% RSLogix 500 project TOFF Que 3.RSS, saved by version 8.30.00.15 %
PROJECT "UNTITLED"    % processor: MicroLogix 1400 %

PROGRAM FILES
  LAD 2   5 rungs

DATA FILES
  O0 OUTPUT  6 elements
  I1 INPUT  8 elements
  S2 STATUS  66 elements
  B3 BINARY  1 elements
  T4 TIMER  3 elements
  C5 COUNTER  1 elements
  R6 CONTROL  1 elements
  N7 INTEGER  1 elements
  F8 FLOAT  1 elements

LADDER 2
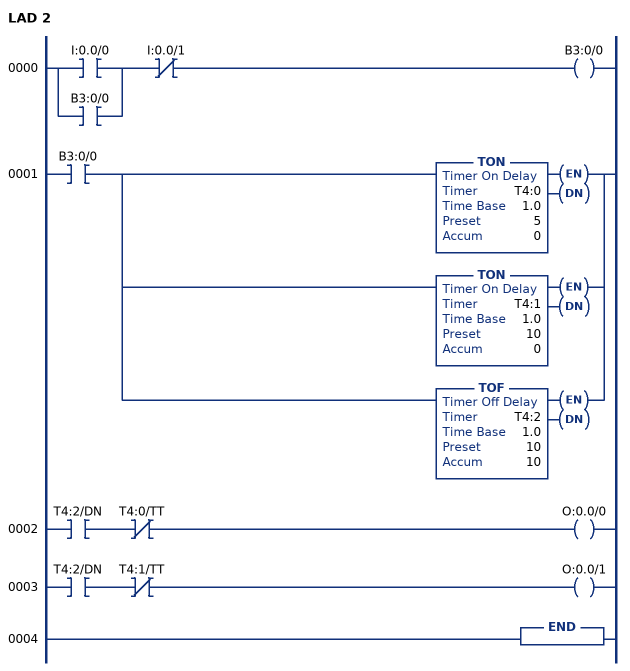
% Rung: 0 %
SOR BST XIC I:0.0/0 NXB XIC B3:0/0 BND XIO I:0.0/1 OTE B3:0/0 EOR
% Rung: 1 %
SOR XIC B3:0/0 BST TON T4:0 1.0 5 0 NXB BST TON T4:1 1.0 10 0 NXB TOF T4:2 1.0 10 10 BND BND EOR
% Rung: 2 %
SOR XIC T4:2/DN XIO T4:0/TT OTE O:0.0/0 EOR
% Rung: 3 %
SOR XIC T4:2/DN XIO T4:1/TT OTE O:0.0/1 EOR
% Rung: 4 %
SOR END EOR

DATA TABLE (non-zero values as saved)
DATA T4
% .PRE .ACC %
% T4:0 % 5 0
% T4:1 % 10 0
% T4:2 % 10 10
